TYPE E_DataExchaSteps :
(
	DATAEXCHA_STATE_IDLE,
	DATAEXCHA_STATE_SEND_START,
	DATAEXCHA_STATE_SEND_WAIT,
	DATAEXCHA_STATE_RECEIVE_START,
	DATAEXCHA_STATE_RECEIVE_WAIT,
	DATAEXCHA_STATE_ERROR
);
END_TYPE

(* stored: Version 1.1.0.1, ProductVersion 3.1.4024.4
   DUT E_DataExchaSteps: Id {efa46226-e271-4357-b9e5-8c37658433ce} *)
